SUBAPPLICATION NMEA_Auswahl (* Waehlt per Button die NMEA2000-Geschwindigkeit ueber Grund (Speed over Ground) als Quelle aus, merkt sich die Auswahl persistent im NVS, setzt bei Auswahl die anderen Quellen zurueck und liefert die NMEA-Sensordaten nach aussen *)
  (* Standard: 61499-2 *)
  (* Version 1.0, 2026-08-27, Franz *)
  PACKAGE FBs::Baumsetzer::func::Automatik;
  IMPORT NVS_Keys::Key_NMEA_Store;
  IMPORT isobus::UT::io::Button::ButtonActivationCode::BT_RELEASED_UNLATCHED;
  IMPORT test::FBs::Baumsetzer::Constants::DefaultPool::Button_NMEA;
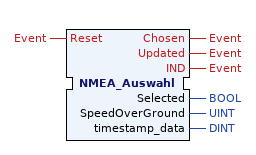
  EVENT_INPUT
    Reset; (* Anforderung von einer der anderen Quellen: eigene Auswahl zuruecksetzen *)
  END_EVENT
  EVENT_OUTPUT
    Chosen; (* Button_NMEA wurde gedrueckt: eigene Auswahl setzen und alle anderen Quellen zuruecksetzen *)
    Updated; (* Ausgewaehlt-Status verfuegbar bzw. geaendert (Init-Lesen oder Aenderung); Trigger fuer nachgelagerte Verarbeitung (u.a. Hintergrundfarbe) *)
    IND; (* Neue NMEA-Daten empfangen (Indication von COGSOGRapidUpdate) *)
  END_EVENT
  VAR_OUTPUT
    Selected : BOOL; (* TRUE wenn NMEA aktuell als Geschwindigkeitsquelle ausgewaehlt ist *)
    SpeedOverGround : UINT; (* Geschwindigkeit ueber Grund aus NMEA2000 COG&SOG Rapid Update (PGN 129026) *)
    timestamp_data : DINT; (* Zeitstempel der letzten NMEA-Botschaft *)
  END_VAR
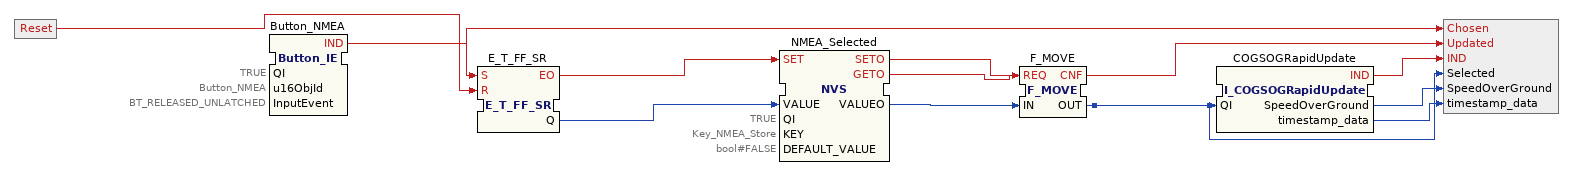
  FBS
    Button_NMEA : isobus::UT::io::Button::Button_IE(QI := TRUE, u16ObjId := Button_NMEA, InputEvent := BT_RELEASED_UNLATCHED);
    E_T_FF_SR : iec61499::events::E_T_FF_SR;
    NMEA_Selected : logiBUS::storage::esp32_nvs::NVS(QI := TRUE, KEY := Key_NMEA_Store, DEFAULT_VALUE := bool#FALSE);
    F_MOVE : iec61131::selection::F_MOVE; {SET_ATTRIBUTE(DataType, BOOL)}
    COGSOGRapidUpdate : isobus::tecu::I_COGSOGRapidUpdate;
  END_FBS
  EVENT_CONNECTIONS
    Button_NMEA.IND TO E_T_FF_SR.S;
    Button_NMEA.IND TO Chosen;
    Reset TO E_T_FF_SR.R;
    E_T_FF_SR.EO TO NMEA_Selected.SET;
    NMEA_Selected.SETO TO F_MOVE.REQ;
    NMEA_Selected.GETO TO F_MOVE.REQ;
    F_MOVE.CNF TO Updated;
    COGSOGRapidUpdate.IND TO IND;
  END_CONNECTIONS
  DATA_CONNECTIONS
    E_T_FF_SR.Q TO NMEA_Selected.VALUE;
    NMEA_Selected.VALUEO TO F_MOVE.IN;
    F_MOVE.OUT TO COGSOGRapidUpdate.QI;
    F_MOVE.OUT TO Selected;
    COGSOGRapidUpdate.SpeedOverGround TO SpeedOverGround;
    COGSOGRapidUpdate.timestamp_data TO timestamp_data;
  END_CONNECTIONS
END_SUBAPPLICATION
